// TIA Portal V17 export
// export: Created 2025-03-07T09:19:30.1038855Z, ExportSetting WithDefaults, DisplayName Totally Integrated Automation Portal, DisplayVersion V17 Update 8, DisplayName TIA Portal Openness, DisplayVersion V17 Update 8, DisplayName TIA Portal Version Control Interface, DisplayVersion V17, DisplayName SINAMICS Startdrive Advanced, DisplayVersion V17 SP2, DisplayName SINAMICS Startdrive G110M, G120, G120C, G120D, G120P, G115D, DisplayVersion V17 SP2, DisplayName SINAMICS Startdrive G130, G150, S120, S150, SINAMICS MV, S210, DisplayVersion V17 SP2, DisplayName STEP 7 Professional, DisplayVersion V17 Update 8, DisplayName SINUMERIK ONE STEP 7 Toolbox, DisplayVersion V17 Update 12, DisplayName SINUMERIK 840D sl STEP 7 Toolbox, DisplayVersion V17 Update 12, DisplayName STEP 7 Safety, DisplayVersion V17 Update 6, DisplayName WinCC Advanced, DisplayVersion V17 Update 8
TYPE "LBP_typeMcp310AdditionalOutput"
TITLE = MCP 310 image / Imagen de MCP 310 / MCP 310 Abbild
// Additional output image of MCP 310 / Imagen de salida adicional de MCP 310 / Zusätzliches Ausgangsabbild von MCP 310
// stored: IsFailsafeCompliant false
   STRUCT
      reserved0 : Byte;
      reserved1 : Byte;
   END_STRUCT;
END_TYPE
